// matB=num*MatA
FUNCTION matMultiNum : BOOL
VAR_IN_OUT CONSTANT
	matA :ARRAY[*,*] OF LREAL;
	num : LREAL;
END_VAR

VAR_IN_OUT 
	matB :ARRAY[*,*] OF LREAL;
END_VAR

VAR
	m,n :DINT;
	i,j, k :DINT;
 
END_VAR

m:=UPPER_BOUND(matB,1);
n:= UPPER_BOUND(matB,2);
FOR i:=1 TO m DO
	FOR j:=1 TO n DO
		matB[i,j]:=num*matA[i,j];
	END_FOR
END_FOR

END_FUNCTION

(* stored: Version 1.1.0.1, ProductVersion 3.1.4024.11
   POU matMultiNum: Id {36ed1c69-32ec-4eea-80af-d1c51a3753b9}, SpecialFunc None *)
